FUNCTION_BLOCK CONNECT_MQTT
  {SET_ATTRIBUTE(OpcUa, POINT.STARTPOINT)}
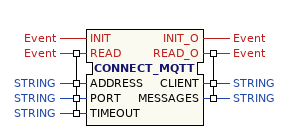
  EVENT_INPUT
    INIT;
    READ WITH ADDRESS, PORT, TIMEOUT;
  END_EVENT
  EVENT_OUTPUT
    INIT_O;
    READ_O WITH CLIENT, MESSAGES;
  END_EVENT
  VAR_INPUT
    ADDRESS : STRING; {SET_ATTRIBUTE(OpcUa, Constant)}
    PORT : STRING; {SET_ATTRIBUTE(OpcUa, Constant)}
    TIMEOUT : STRING; {SET_ATTRIBUTE(OpcUa, Constant)}
  END_VAR
  VAR_OUTPUT
    CLIENT : STRING; {SET_ATTRIBUTE(OpcUa, Variable)}
    MESSAGES : STRING; {SET_ATTRIBUTE(OpcUa, Variable)}
  END_VAR
END_FUNCTION_BLOCK
